(* IEC 61131-3 sources: POMIRTS_lab3/AS/Library/AsIOAcc, 3 files *)

(* ---- AsIOAcc.typ ---- *)
(********************************************************************
 * COPYRIGHT -- Bernecker + Rainer
 ********************************************************************
 * Library: AsIOAcc
 * File: AsIOAcc.typ
 * Author: B+R
 ********************************************************************
 * Data types of library AsIOAcc
 ********************************************************************)

TYPE
	IOAC_I_TYPE : STRUCT			(*internal use*)
		StateMan	: UINT ;
		ErrMan	: UINT ;
		Init	: UDINT ;
		Taskhandle	: UDINT ;
		Semaphore	: UDINT ;
		Requestsize	: UDINT ;
		Answersize	: UDINT ;
		pAccessObj	: UDINT ;
		Offset	: UDINT ;
		flags	: UDINT ;
	END_STRUCT;
END_TYPE

(* ---- AsIOAcc.fun ---- *)
(********************************************************************
 * COPYRIGHT -- Bernecker + Rainer
 ********************************************************************
 * Library: AsIOAcc
 * File: AsIOAcc.fun
 * Author: B+R
 ********************************************************************
 * Functions and function blocks of library AsIOAcc
 ********************************************************************)

FUNCTION_BLOCK AsIOAccRead				(*reads noncyclical register (only inputs); asynchronous execution*)
	VAR_INPUT
		enable	:BOOL;					(*enables execution*)
		pDeviceName	:UDINT;				(*device name given as a pointer*)
		pChannelName	:UDINT;			(*pointer to the channel name*)
	END_VAR
	VAR_OUTPUT
		status	:UINT;					(*execution status: ERR_OK, ERR_FUB_ENABLE_FALSE, ERR_FUB_BUSY, 0xXXXX = see help*)
		value	:UDINT;					(*value read*)
	END_VAR
	VAR
		intern	:IOAC_I_TYPE;			(*internal variable*)
	END_VAR
END_FUNCTION_BLOCK

FUNCTION_BLOCK AsIOAccWrite				(*writes noncyclical register (ONLY outputs); asynchronous execution*)
	VAR_INPUT
		enable	:BOOL;					(*enables execution*)
		pDeviceName	:UDINT;				(*device name given as a pointer*)
		pChannelName	:UDINT;			(*pointer to the channel name*)
		value	:UDINT;					(*value to be written*)
	END_VAR
	VAR_OUTPUT
		status	:UINT;					(*execution status: ERR_OK, ERR_FUB_ENABLE_FALSE, ERR_FUB_BUSY, 0xXXXX = see help*)
	END_VAR
	VAR
		intern	:IOAC_I_TYPE;			(*internal variable*)
	END_VAR
END_FUNCTION_BLOCK

FUNCTION_BLOCK AsIOAccReadReg
	VAR_INPUT
		enable			: BOOL;			(*enables execution*)
		nodeNr			: USINT;		(*node number of x2x module*)
		registerNr		: UINT;			(*register number*)
		size			: USINT;		(*register size*)
	END_VAR

	VAR_OUTPUT
		status			: UINT;			(*execution status: ERR_OK, ERR_FUB_ENABLE_FALSE, ERR_FUB_BUSY, 0xXXXX = see help*)
		value			: UDINT;		(*regsiter value*)
	END_VAR

	VAR
        i_state			: UINT;			(*internal variable*)
		i_result		: UINT;			(*internal variable*)
        i_tmp			: UDINT;		(*internal variable*)
	END_VAR
END_FUNCTION_BLOCK

FUNCTION_BLOCK AsIOAccWriteReg
	VAR_INPUT
		enable			: BOOL;			(*enables execution*)
		nodeNr			: USINT;		(*node number of x2x module*)
		registerNr		: UINT;			(*register number*)
		size			: USINT;		(*register size*)
		value			: UDINT;		(*new register value*)
	END_VAR

	VAR_OUTPUT
		status			: UINT;			(*execution status: ERR_OK, ERR_FUB_ENABLE_FALSE, ERR_FUB_BUSY, 0xXXXX = see help*)
	END_VAR

	VAR
        i_state			: UINT;			(*internal variable*)
		i_result		: UINT;			(*internal variable*)
        i_tmp			: UDINT;		(*internal variable*)
	END_VAR
END_FUNCTION_BLOCK

(* ---- AsIOAcc.var ---- *)
(********************************************************************
 * COPYRIGHT -- Bernecker + Rainer
 ********************************************************************
 * Library: AsIOAcc
 * File: AsIOAcc.var
 * Author: B+R
 ********************************************************************
 * Local variables of library AsIOAcc
 ********************************************************************)

VAR CONSTANT
	ioacERR_INTERNAL        : UINT := 30190;		(*internal error*)
	ioacERR_DEVICE          : UINT := 30191;		(*I/O module does not exist*)
	ioacERR_CHANNEL         : UINT := 30192;		(*incorrect channel name specified*)
	ioacERR_TIMEOUT         : UINT := 30193;		(*timeout reached*)
	ioacERR_NOTSUPPORTED    : UINT := 30194;		(*not supported*)
	ioacERR_PARAMETER		: UINT := 30195;		(*invalid parameter*)
	ioacERR_ACCESS			: UINT := 30196;		(*access error*)
END_VAR
